PROGRAM MAIN
VAR
	RawNumber		:LREAL := 2.56870000002;
	DecimalPlaces	:USINT := 3;
	RoundedNumber	:LREAL;
	RoundedNumber_m2	:LREAL;
END_VAR

RoundedNumber := fnRoundLREAL(RawNumber, DecimalPlaces);
RoundedNumber_m2 := fnRoundLREAL(RawNumber, DecimalPlaces);

END_PROGRAM

(* stored: Version 1.1.0.1, ProductVersion 3.1.4024.16
   POU MAIN: Id {9c6917e1-7882-4283-8684-162549e06f53}, SpecialFunc None *)
